ABB RobotStudio station: Project2.rsstnx

Station Project2 (saved by RobotStudio 22.3.10141.1)
Controller Controlador1
  mechanical unit ROB_1: IRB910SC_3_45__01, 4 joints, base frame (0, 0, 0) mm
  mechanical unit ROB_2: IRB1600_6_120__02, 6 joints, base frame (1000, 0, 0) mm
  mechanical unit ROB_3: IRB1600_10_120__01, 6 joints, base frame (0, 1000, 0) mm
Layout (positions relative to the parent item):
  - IRB910SC_3_45__01 [mechanism, from Robots\IRB910SC_3_45__01.rslib] at (0, 0, 0) mm; joint values [0, 0, 0, 0] (rad or m)
  - IRB1600_6_120__02 [mechanism, from Robots\IRB1600_6_120_G_02.rslib] at (1000, 0, 0) mm; joint values [0, 0, 0, 0, 0.5236, 0] (rad or m)
  - IRB1600_10_120__01 [mechanism, from Robots\IRB1600_10_120_G_01.rslib] at (0, 1000, 0) mm; joint values [0, 0, 0, 0, 0.5236, 0] (rad or m)
  - Fence_2500 [graphiccomponentgroup, from Equipment\Fence_2500.rslib] at (2000, 0, 0) mm
    - Body 1 [part, from Equipment\Fence_2500.rslib]
    - Body 2 [part, from Equipment\Fence_2500.rslib]
